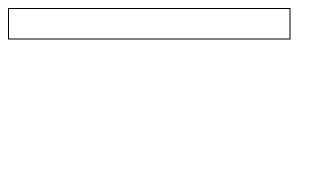
[picture p24: P60013 (HMI screen)]
rectangle at (270,210)-(321,241): text "ESC"
rectangle at (270,210)-(321,241): text "ESC"; invisible if NOT.alarm
rectangle at (20,80)-(302,111): text "Band Brake Limit:"
rectangle at (20,120)-(302,151): text "Water Brake Limit:"
rectangle at (200,80)-(301,111): text "%s %%"; shows bandLimit; invisible if editMode
rectangle at (200,120)-(301,151): text "%s %%"; shows wcbLimit
*)

(* Visualisation START_PAGE/MAIN_MANU/MAIN_MENU_1/DISPLAY_SETUP/1_DISPLAY_SETUP/2_Set_Water_Brake_Limit/P60014
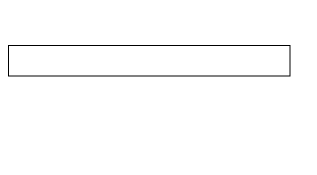
rectangle at (270,210)-(321,241): text "ESC"
rectangle at (270,210)-(321,241): text "ESC"; invisible if NOT.alarm
rectangle at (20,80)-(302,111): text "Band Brake Limit:"
rectangle at (20,120)-(302,151): text "Water Brake Limit:"
rectangle at (200,80)-(301,111): text "%s %%"; shows bandLimit
rectangle at (200,120)-(301,151): text "%s %%"; shows wcbLimit; invisible if editMode
*)

(* Visualisation START_PAGE/MAIN_MANU/MAIN_MENU_1/DISPLAY_SETUP/1_DISPLAY_SETUP/P65000
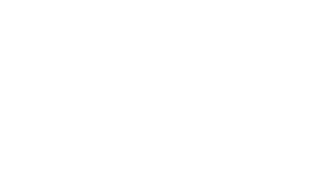
rectangle at (20,120)-(302,151): text "Water Brake Limit:"; alarm colour if SELECT_PAGE.MenuItem=2
rectangle at (20,80)-(302,111): text "Band Brake Limit:"; alarm colour if SELECT_PAGE.MenuItem=1
rectangle at (270,210)-(321,241): text "ESC"
rectangle at (270,210)-(321,241): text "ESC"; invisible if NOT.alarm
rectangle at (200,80)-(301,111): text "%s %%"; shows bandLimit
rectangle at (200,120)-(301,151): text "%s %%"; shows wcbLimit
*)
